PROGRAM PRG_ScrewdriverManager
VAR
    fbScrewdriver1 : FB_ScrewdriverControl;
    fbScrewdriver2 : FB_ScrewdriverControl;
END_VAR

// 两个运行实例共用同一FB类型，但端口、缓存、状态机和定时器完全独立。
// 上层FB_DualScrewdriverAction只通过两个GVL接口组合同步工艺条件。
fbScrewdriver1(
    bEnable := GVL_Screwdriver.bEnableScrewdriver1,
    ioScrewdriver := GVL_Screwdriver.stScrewdriver1
);

fbScrewdriver2(
    bEnable := GVL_Screwdriver.bEnableScrewdriver2,
    ioScrewdriver := GVL_Screwdriver.stScrewdriver2
);

END_PROGRAM

(* stored: Version 1.1.0.1, ProductVersion 3.1.4026.20
   POU PRG_ScrewdriverManager: Id {931F1626-2951-4BD0-B3A5-31A71020D522}, SpecialFunc None *)
